PROGRAM SkillSet
VAR
	Move_2P2			:Skill_Position_anfahren;
	Grip_2P2			:Skill_Greifer_Pos_Anfahren;
END_VAR

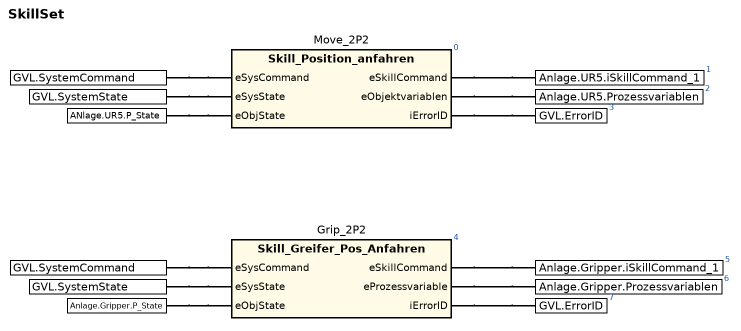
Move_2P2(eSysCommand := GVL.SystemCommand, eSysState := GVL.SystemState, eObjState := ANlage.UR5.P_State); // Skill_Position_anfahren
Anlage.UR5.iSkillCommand_1 := Move_2P2.eSkillCommand;
Anlage.UR5.Prozessvariablen := Move_2P2.eObjektvariablen;
GVL.ErrorID := Move_2P2.iErrorID;
Grip_2P2(eSysCommand := GVL.SystemCommand, eSysState := GVL.SystemState, eObjState := Anlage.Gripper.P_State); // Skill_Greifer_Pos_Anfahren
Anlage.Gripper.iSkillCommand_1 := Grip_2P2.eSkillCommand;
Anlage.Gripper.Prozessvariablen := Grip_2P2.eProzessvariable;
GVL.ErrorID := Grip_2P2.iErrorID;

END_PROGRAM

(* stored: Version 1.1.0.1
   POU SkillSet: Id {ae96e4ed-6c2f-4080-bbe5-bf79d7c4e711}, SpecialFunc None *)
